(* CODESYS project Exp_1.project
   Company: ifm electronic
   Description: Project template with CR711S configured 2.25MByte Standard 2.25MByte Safety
   Title: ifmCR711S_TemplateProject
   Version: 2.4.10.0

Project tree, tasks and I/O mapping:
  SafetyPLC : CR711S SIL2, ifm electronic, order no. CR711S, version 3.2.0.0
    application Application
      libraries: ifmR360-3, * (ifm electronic)
      task Task (cyclic, interval t#10ms, priority 1, watchdog t#8ms x 1) calls PLC_PRG
      global variables EVL
      program PLC_PRG [ST]
    Communication : Communication, ifm electronic, version 3.2.0.0
      CAN : CAN, ifm electronic, version 3.2.0.0
      Ethernet : Ethernet, ifm electronic, version 3.2.0.0
    HMI : HMI, ifm electronic, version 3.2.0.0
      User_LEDs : User_LEDs, ifm electronic, version 3.2.0.0
          input  UserLED0_I : LED_IEC_B_INPUT_MAPPING_TYPE  // UserLED0_I
          input  UserLED1_I : LED_IEC_B_INPUT_MAPPING_TYPE  // UserLED1_I
          input  UserLED2_I : LED_IEC_B_INPUT_MAPPING_TYPE  // UserLED2_I
          input  UserLED3_I : LED_IEC_B_INPUT_MAPPING_TYPE  // UserLED3_I
          output UserLED0_Q : LED_IEC_B_OUTPUT_MAPPING_TYPE  // User LED 0
          output UserLED1_Q : LED_IEC_B_OUTPUT_MAPPING_TYPE  // User LED 1
          output UserLED2_Q : LED_IEC_B_OUTPUT_MAPPING_TYPE  // User LED 2
          output UserLED3_Q : LED_IEC_B_OUTPUT_MAPPING_TYPE  // User LED 3
    Local_IO : Local_IO, ifm electronic, version 3.2.0.0
      Inputs : Inputs, ifm electronic, version 3.2.0.0
          input  IN0100_I : IN_MULTIFUNCTION_A_INPUT_MAPPING_TYPE  // IN0100_I
          input  IN0101_I : IN_MULTIFUNCTION_A_INPUT_MAPPING_TYPE  // IN0101_I
          input  IN0102_I : IN_MULTIFUNCTION_A_INPUT_MAPPING_TYPE  // IN0102_I
          input  IN0103_I : IN_MULTIFUNCTION_A_INPUT_MAPPING_TYPE  // IN0103_I
          input  IN0200_I : IN_MULTIFUNCTION_A_INPUT_MAPPING_TYPE  // IN0200_I
          input  IN0201_I : IN_MULTIFUNCTION_A_INPUT_MAPPING_TYPE  // IN0201_I
          input  IN0202_I : IN_MULTIFUNCTION_A_INPUT_MAPPING_TYPE  // IN0202_I
          input  IN0203_I : IN_MULTIFUNCTION_A_INPUT_MAPPING_TYPE  // IN0203_I
          input  IN0600_I : IN_MULTIFUNCTION_A_INPUT_MAPPING_TYPE  // IN0600_I
          input  IN0601_I : IN_MULTIFUNCTION_A_INPUT_MAPPING_TYPE  // IN0601_I
          input  IN0602_I : IN_MULTIFUNCTION_A_INPUT_MAPPING_TYPE  // IN0602_I
          input  IN0603_I : IN_MULTIFUNCTION_A_INPUT_MAPPING_TYPE  // IN0603_I
          input  IN0700_I : IN_MULTIFUNCTION_A_INPUT_MAPPING_TYPE  // IN0700_I
          input  IN0701_I : IN_MULTIFUNCTION_A_INPUT_MAPPING_TYPE  // IN0701_I
          input  IN0702_I : IN_MULTIFUNCTION_A_INPUT_MAPPING_TYPE  // IN0702_I
          input  IN0703_I : IN_MULTIFUNCTION_A_INPUT_MAPPING_TYPE  // IN0703_I
          input  IN0400_I : IN_RESISTOR_A_INPUT_MAPPING_TYPE  // IN0400_I
          input  IN0401_I : IN_RESISTOR_A_INPUT_MAPPING_TYPE  // IN0401_I
          input  IN0900_I : IN_RESISTOR_A_INPUT_MAPPING_TYPE  // IN0900_I
          input  IN0901_I : IN_RESISTOR_A_INPUT_MAPPING_TYPE  // IN0901_I
          input  IN0300_I : IN_DIGITAL_B_INPUT_MAPPING_TYPE  // IN0300_I
          input  IN0301_I : IN_DIGITAL_B_INPUT_MAPPING_TYPE  // IN0301_I
          input  IN0800_I : IN_DIGITAL_B_INPUT_MAPPING_TYPE  // IN0800_I
          input  IN0801_I : IN_DIGITAL_B_INPUT_MAPPING_TYPE  // IN0801_I
          input  COM_RESET_I : IN_COMMUNICATION_RESET_INPUT_MAPPING_TYPE  // COM_RESET_I
          input  IN0000_I : IN_FREQUENCY_B_CHANNEL_A_INPUT_MAPPING_TYPE  // IN0000_I
          input  IN0002_I : IN_FREQUENCY_B_CHANNEL_A_INPUT_MAPPING_TYPE  // IN0002_I
          input  IN0500_I : IN_FREQUENCY_B_CHANNEL_A_INPUT_MAPPING_TYPE  // IN0500_I
          input  IN0502_I : IN_FREQUENCY_B_CHANNEL_A_INPUT_MAPPING_TYPE  // IN0502_I
          input  IN0001_I : IN_FREQUENCY_B_CHANNEL_B_INPUT_MAPPING_TYPE  // IN0001_I
          input  IN0003_I : IN_FREQUENCY_B_CHANNEL_B_INPUT_MAPPING_TYPE  // IN0003_I
          input  IN0501_I : IN_FREQUENCY_B_CHANNEL_B_INPUT_MAPPING_TYPE  // IN0501_I
          input  IN0503_I : IN_FREQUENCY_B_CHANNEL_B_INPUT_MAPPING_TYPE  // IN0503_I
      Outputs : Outputs, ifm electronic, version 3.2.0.0
          input  OUT0006_I : OUT_PWM_40_BRIDGE_A_INPUT_MAPPING_TYPE  // OUT0006_I
          input  OUT0106_I : OUT_PWM_40_BRIDGE_A_INPUT_MAPPING_TYPE  // OUT0106_I
          input  OUT0206_I : OUT_PWM_40_BRIDGE_A_INPUT_MAPPING_TYPE  // OUT0206_I
          input  OUT0008_I : OUT_PWM_40_A_INPUT_MAPPING_TYPE  // OUT0008_I
          input  OUT0108_I : OUT_PWM_40_A_INPUT_MAPPING_TYPE  // OUT0108_I
          input  OUT0208_I : OUT_PWM_40_A_INPUT_MAPPING_TYPE  // OUT0208_I
          input  OUT0000_I : OUT_PWM_25_A_INPUT_MAPPING_TYPE  // OUT0000_I
          input  OUT0002_I : OUT_PWM_25_A_INPUT_MAPPING_TYPE  // OUT0002_I
          input  OUT0004_I : OUT_PWM_25_A_INPUT_MAPPING_TYPE  // OUT0004_I
          input  OUT0100_I : OUT_PWM_25_A_INPUT_MAPPING_TYPE  // OUT0100_I
          input  OUT0102_I : OUT_PWM_25_A_INPUT_MAPPING_TYPE  // OUT0102_I
          input  OUT0104_I : OUT_PWM_25_A_INPUT_MAPPING_TYPE  // OUT0104_I
          input  OUT0200_I : OUT_PWM_25_A_INPUT_MAPPING_TYPE  // OUT0200_I
          input  OUT0202_I : OUT_PWM_25_A_INPUT_MAPPING_TYPE  // OUT0202_I
          input  OUT0204_I : OUT_PWM_25_A_INPUT_MAPPING_TYPE  // OUT0204_I
          input  OUT3001_I : OUT_VOLTAGE_A_INPUT_MAPPING_TYPE  // OUT3001_I
          input  OUT3000_I : OUT_SUPPLY_A_INPUT_MAPPING_TYPE  // OUT3000_I
          input  OUT0001_I : OUT_PWM_25_B_INPUT_MAPPING_TYPE  // OUT0001_I
          input  OUT0003_I : OUT_PWM_25_B_INPUT_MAPPING_TYPE  // OUT0003_I
          input  OUT0005_I : OUT_PWM_25_B_INPUT_MAPPING_TYPE  // OUT0005_I
          input  OUT0101_I : OUT_PWM_25_B_INPUT_MAPPING_TYPE  // OUT0101_I
          input  OUT0103_I : OUT_PWM_25_B_INPUT_MAPPING_TYPE  // OUT0103_I
          input  OUT0105_I : OUT_PWM_25_B_INPUT_MAPPING_TYPE  // OUT0105_I
          input  OUT0201_I : OUT_PWM_25_B_INPUT_MAPPING_TYPE  // OUT0201_I
          input  OUT0203_I : OUT_PWM_25_B_INPUT_MAPPING_TYPE  // OUT0203_I
          input  OUT0205_I : OUT_PWM_25_B_INPUT_MAPPING_TYPE  // OUT0205_I
          input  OUT0007_I : OUT_PWM_40_BRIDGE_A_INPUT_MAPPING_TYPE  // OUT0007_I
          input  OUT0107_I : OUT_PWM_40_BRIDGE_A_INPUT_MAPPING_TYPE  // OUT0107_I
          input  OUT0207_I : OUT_PWM_40_BRIDGE_A_INPUT_MAPPING_TYPE  // OUT0207_I
          output OUT0006_Q : OUT_PWM_40_BRIDGE_A_OUTPUT_MAPPING_TYPE  // OUT0006_Q
          output OUT0106_Q : OUT_PWM_40_BRIDGE_A_OUTPUT_MAPPING_TYPE  // OUT0106_Q
          output OUT0206_Q : OUT_PWM_40_BRIDGE_A_OUTPUT_MAPPING_TYPE  // OUT0206_Q
          output OUT0008_Q : OUT_PWM_40_A_OUTPUT_MAPPING_TYPE  // OUT0008_Q
          output OUT0108_Q : OUT_PWM_40_A_OUTPUT_MAPPING_TYPE  // OUT0108_Q
          output OUT0208_Q : OUT_PWM_40_A_OUTPUT_MAPPING_TYPE  // OUT0208_Q
          output OUT0000_Q : OUT_PWM_25_A_OUTPUT_MAPPING_TYPE  // OUT0000_Q
          output OUT0002_Q : OUT_PWM_25_A_OUTPUT_MAPPING_TYPE  // OUT0002_Q
          output OUT0004_Q : OUT_PWM_25_A_OUTPUT_MAPPING_TYPE  // OUT0004_Q
          output OUT0100_Q : OUT_PWM_25_A_OUTPUT_MAPPING_TYPE  // OUT0100_Q
          output OUT0102_Q : OUT_PWM_25_A_OUTPUT_MAPPING_TYPE  // OUT0102_Q
          output OUT0104_Q : OUT_PWM_25_A_OUTPUT_MAPPING_TYPE  // OUT0104_Q
          output OUT0200_Q : OUT_PWM_25_A_OUTPUT_MAPPING_TYPE  // OUT0200_Q
          output OUT0202_Q : OUT_PWM_25_A_OUTPUT_MAPPING_TYPE  // OUT0202_Q
          output OUT0204_Q : OUT_PWM_25_A_OUTPUT_MAPPING_TYPE  // OUT0204_Q
          output OUT3001_Q : OUT_VOLTAGE_A_OUTPUT_MAPPING_TYPE  // OUT3001_Q
          output OUT3000_Q : OUT_SUPPLY_A_OUTPUT_MAPPING_TYPE  // OUT3000_Q
          output OUT0001_Q : OUT_PWM_25_B_OUTPUT_MAPPING_TYPE  // OUT0001_Q
          output OUT0003_Q : OUT_PWM_25_B_OUTPUT_MAPPING_TYPE  // OUT0003_Q
          output OUT0005_Q : OUT_PWM_25_B_OUTPUT_MAPPING_TYPE  // OUT0005_Q
          output OUT0101_Q : OUT_PWM_25_B_OUTPUT_MAPPING_TYPE  // OUT0101_Q
          output OUT0103_Q : OUT_PWM_25_B_OUTPUT_MAPPING_TYPE  // OUT0103_Q
          output OUT0105_Q : OUT_PWM_25_B_OUTPUT_MAPPING_TYPE  // OUT0105_Q
          output OUT0201_Q : OUT_PWM_25_B_OUTPUT_MAPPING_TYPE  // OUT0201_Q
          output OUT0203_Q : OUT_PWM_25_B_OUTPUT_MAPPING_TYPE  // OUT0203_Q
          output OUT0205_Q : OUT_PWM_25_B_OUTPUT_MAPPING_TYPE  // OUT0205_Q
          output OUT0007_Q : OUT_PWM_40_BRIDGE_A_OUTPUT_MAPPING_TYPE  // OUT0007_Q
          output OUT0107_Q : OUT_PWM_40_BRIDGE_A_OUTPUT_MAPPING_TYPE  // OUT0107_Q
          output OUT0207_Q : OUT_PWM_40_BRIDGE_A_OUTPUT_MAPPING_TYPE  // OUT0207_Q
      System_Inputs : System_Inputs, ifm electronic, version 3.2.0.0
          input  VBB30 : IN_SYSTEM_VOLTAGE_INPUT_MAPPING_TYPE  // VBB30
          input  VBB15 : IN_SYSTEM_VOLTAGE_INPUT_MAPPING_TYPE  // VBB15
          input  TemperatureBoard0 : IN_TEMPERATURE_INPUT_MAPPING_TYPE  // TemperatureBoard0
          input  TemperatureChip0 : IN_TEMPERATURE_INPUT_MAPPING_TYPE  // TemperatureChip0
      System_Outputs : System_Outputs, ifm electronic, version 3.2.0.0
          input  VBB0_SW_I : OUT_GROUP_SWITCH_INPUT_MAPPING_TYPE  // VBB0_SW_I
          input  VBB1_SW_I : OUT_GROUP_SWITCH_INPUT_MAPPING_TYPE  // VBB1_SW_I
          input  VBB2_SW_I : OUT_GROUP_SWITCH_INPUT_MAPPING_TYPE  // VBB2_SW_I
          output VBB0_SW_Q : OUT_GROUP_SWITCH_OUTPUT_MAPPING_TYPE  // VBB0_SW_Q
          output VBB1_SW_Q : OUT_GROUP_SWITCH_OUTPUT_MAPPING_TYPE  // VBB1_SW_Q
          output VBB2_SW_Q : OUT_GROUP_SWITCH_OUTPUT_MAPPING_TYPE  // VBB2_SW_Q
          output SUPPLY_SWITCH_Q : OUT_SYS_SWITCH_OUTPUT_MAPPING_TYPE  // SUPPLY_SWITCH_Q
  StandardPLC : CR711S Standard, ifm electronic, order no. CR711S, version 3.2.0.0
    application Application
      libraries: ifmR360-3, 1.1.1.0 (ifm electronic); Util, * (System); Standard, * (System); CR711S IOWrapper, 1.0.4.9 (ifm electronic)
      task Task (cyclic, interval t#10ms, priority 0) calls PLC_PRG
      EVC
      program PLC_PRG [ST]
      program CR711S_Config [ST]: config_inputs, config_outgroups, config_outputs
      program CAN_INIT [ST]
      program CA_TX [FBD]
      program CAN_RX [FBD]
    Communication : Communication, ifm electronic, version 3.2.0.0
      CAN : CAN, ifm electronic, version 3.2.0.0
      Ethernet : Ethernet, ifm electronic, version 3.2.0.0
    HMI : HMI, ifm electronic, version 3.2.0.0
      User_LEDs : User_LEDs, ifm electronic, version 3.2.0.0
          input  UserLED0_I : LED_IEC_B_INPUT_MAPPING_TYPE  // UserLED0_I
          input  UserLED1_I : LED_IEC_B_INPUT_MAPPING_TYPE  // UserLED1_I
          input  UserLED2_I : LED_IEC_B_INPUT_MAPPING_TYPE  // UserLED2_I
          input  UserLED3_I : LED_IEC_B_INPUT_MAPPING_TYPE  // UserLED3_I
          output UserLED0_Q : LED_IEC_B_OUTPUT_MAPPING_TYPE  // User LED 0
          output UserLED1_Q : LED_IEC_B_OUTPUT_MAPPING_TYPE  // User LED 1
          output UserLED2_Q : LED_IEC_B_OUTPUT_MAPPING_TYPE  // User LED 2
          output UserLED3_Q : LED_IEC_B_OUTPUT_MAPPING_TYPE  // User LED 3
    Local_IO : Local_IO, ifm electronic, version 3.2.0.0
      Inputs : Inputs, ifm electronic, version 3.2.0.0
          input  IN0100_I : IN_MULTIFUNCTION_A_INPUT_MAPPING_TYPE  // IN0100_I
          input  IN0101_I : IN_MULTIFUNCTION_A_INPUT_MAPPING_TYPE  // IN0101_I
          input  IN0102_I : IN_MULTIFUNCTION_A_INPUT_MAPPING_TYPE  // IN0102_I
          input  IN0103_I : IN_MULTIFUNCTION_A_INPUT_MAPPING_TYPE  // IN0103_I
          input  IN0200_I : IN_MULTIFUNCTION_A_INPUT_MAPPING_TYPE  // IN0200_I
          input  IN0201_I : IN_MULTIFUNCTION_A_INPUT_MAPPING_TYPE  // IN0201_I
          input  IN0202_I : IN_MULTIFUNCTION_A_INPUT_MAPPING_TYPE  // IN0202_I
          input  IN0203_I : IN_MULTIFUNCTION_A_INPUT_MAPPING_TYPE  // IN0203_I
          input  IN0600_I : IN_MULTIFUNCTION_A_INPUT_MAPPING_TYPE  // IN0600_I
          input  IN0601_I : IN_MULTIFUNCTION_A_INPUT_MAPPING_TYPE  // IN0601_I
          input  IN0602_I : IN_MULTIFUNCTION_A_INPUT_MAPPING_TYPE  // IN0602_I
          input  IN0603_I : IN_MULTIFUNCTION_A_INPUT_MAPPING_TYPE  // IN0603_I
          input  IN0700_I : IN_MULTIFUNCTION_A_INPUT_MAPPING_TYPE  // IN0700_I
          input  IN0701_I : IN_MULTIFUNCTION_A_INPUT_MAPPING_TYPE  // IN0701_I
          input  IN0702_I : IN_MULTIFUNCTION_A_INPUT_MAPPING_TYPE  // IN0702_I
          input  IN0703_I : IN_MULTIFUNCTION_A_INPUT_MAPPING_TYPE  // IN0703_I
          input  IN0400_I : IN_RESISTOR_A_INPUT_MAPPING_TYPE  // IN0400_I
          input  IN0401_I : IN_RESISTOR_A_INPUT_MAPPING_TYPE  // IN0401_I
          input  IN0900_I : IN_RESISTOR_A_INPUT_MAPPING_TYPE  // IN0900_I
          input  IN0901_I : IN_RESISTOR_A_INPUT_MAPPING_TYPE  // IN0901_I
          input  IN0300_I : IN_DIGITAL_B_INPUT_MAPPING_TYPE  // IN0300_I
          input  IN0301_I : IN_DIGITAL_B_INPUT_MAPPING_TYPE  // IN0301_I
          input  IN0800_I : IN_DIGITAL_B_INPUT_MAPPING_TYPE  // IN0800_I
          input  IN0801_I : IN_DIGITAL_B_INPUT_MAPPING_TYPE  // IN0801_I
          input  COM_RESET_I : IN_COMMUNICATION_RESET_INPUT_MAPPING_TYPE  // COM_RESET_I
          input  IN0000_I : IN_FREQUENCY_B_CHANNEL_A_INPUT_MAPPING_TYPE  // IN0000_I
          input  IN0002_I : IN_FREQUENCY_B_CHANNEL_A_INPUT_MAPPING_TYPE  // IN0002_I
          input  IN0500_I : IN_FREQUENCY_B_CHANNEL_A_INPUT_MAPPING_TYPE  // IN0500_I
          input  IN0502_I : IN_FREQUENCY_B_CHANNEL_A_INPUT_MAPPING_TYPE  // IN0502_I
          input  IN0001_I : IN_FREQUENCY_B_CHANNEL_B_INPUT_MAPPING_TYPE  // IN0001_I
          input  IN0003_I : IN_FREQUENCY_B_CHANNEL_B_INPUT_MAPPING_TYPE  // IN0003_I
          input  IN0501_I : IN_FREQUENCY_B_CHANNEL_B_INPUT_MAPPING_TYPE  // IN0501_I
          input  IN0503_I : IN_FREQUENCY_B_CHANNEL_B_INPUT_MAPPING_TYPE  // IN0503_I
      Outputs : Outputs, ifm electronic, version 3.2.0.0
          input  OUT0006_I : OUT_PWM_40_BRIDGE_A_INPUT_MAPPING_TYPE  // OUT0006_I
          input  OUT0106_I : OUT_PWM_40_BRIDGE_A_INPUT_MAPPING_TYPE  // OUT0106_I
          input  OUT0206_I : OUT_PWM_40_BRIDGE_A_INPUT_MAPPING_TYPE  // OUT0206_I
          input  OUT0008_I : OUT_PWM_40_A_INPUT_MAPPING_TYPE  // OUT0008_I
          input  OUT0108_I : OUT_PWM_40_A_INPUT_MAPPING_TYPE  // OUT0108_I
          input  OUT0208_I : OUT_PWM_40_A_INPUT_MAPPING_TYPE  // OUT0208_I
          input  OUT0000_I : OUT_PWM_25_A_INPUT_MAPPING_TYPE  // OUT0000_I
          input  OUT0002_I : OUT_PWM_25_A_INPUT_MAPPING_TYPE  // OUT0002_I
          input  OUT0004_I : OUT_PWM_25_A_INPUT_MAPPING_TYPE  // OUT0004_I
          input  OUT0100_I : OUT_PWM_25_A_INPUT_MAPPING_TYPE  // OUT0100_I
          input  OUT0102_I : OUT_PWM_25_A_INPUT_MAPPING_TYPE  // OUT0102_I
          input  OUT0104_I : OUT_PWM_25_A_INPUT_MAPPING_TYPE  // OUT0104_I
          input  OUT0200_I : OUT_PWM_25_A_INPUT_MAPPING_TYPE  // OUT0200_I
          input  OUT0202_I : OUT_PWM_25_A_INPUT_MAPPING_TYPE  // OUT0202_I
          input  OUT0204_I : OUT_PWM_25_A_INPUT_MAPPING_TYPE  // OUT0204_I
          input  OUT3001_I : OUT_VOLTAGE_A_INPUT_MAPPING_TYPE  // OUT3001_I
          input  OUT3000_I : OUT_SUPPLY_A_INPUT_MAPPING_TYPE  // OUT3000_I
          input  OUT0001_I : OUT_PWM_25_B_INPUT_MAPPING_TYPE  // OUT0001_I
          input  OUT0003_I : OUT_PWM_25_B_INPUT_MAPPING_TYPE  // OUT0003_I
          input  OUT0005_I : OUT_PWM_25_B_INPUT_MAPPING_TYPE  // OUT0005_I
          input  OUT0101_I : OUT_PWM_25_B_INPUT_MAPPING_TYPE  // OUT0101_I
          input  OUT0103_I : OUT_PWM_25_B_INPUT_MAPPING_TYPE  // OUT0103_I
          input  OUT0105_I : OUT_PWM_25_B_INPUT_MAPPING_TYPE  // OUT0105_I
          input  OUT0201_I : OUT_PWM_25_B_INPUT_MAPPING_TYPE  // OUT0201_I
          input  OUT0203_I : OUT_PWM_25_B_INPUT_MAPPING_TYPE  // OUT0203_I
          input  OUT0205_I : OUT_PWM_25_B_INPUT_MAPPING_TYPE  // OUT0205_I
          input  OUT0007_I : OUT_PWM_40_BRIDGE_A_INPUT_MAPPING_TYPE  // OUT0007_I
          input  OUT0107_I : OUT_PWM_40_BRIDGE_A_INPUT_MAPPING_TYPE  // OUT0107_I
          input  OUT0207_I : OUT_PWM_40_BRIDGE_A_INPUT_MAPPING_TYPE  // OUT0207_I
          output OUT0006_Q : OUT_PWM_40_BRIDGE_A_OUTPUT_MAPPING_TYPE  // OUT0006_Q
          output OUT0106_Q : OUT_PWM_40_BRIDGE_A_OUTPUT_MAPPING_TYPE  // OUT0106_Q
          output OUT0206_Q : OUT_PWM_40_BRIDGE_A_OUTPUT_MAPPING_TYPE  // OUT0206_Q
          output OUT0008_Q : OUT_PWM_40_A_OUTPUT_MAPPING_TYPE  // OUT0008_Q
          output OUT0108_Q : OUT_PWM_40_A_OUTPUT_MAPPING_TYPE  // OUT0108_Q
          output OUT0208_Q : OUT_PWM_40_A_OUTPUT_MAPPING_TYPE  // OUT0208_Q
          output OUT0000_Q : OUT_PWM_25_A_OUTPUT_MAPPING_TYPE  // OUT0000_Q
          output OUT0002_Q : OUT_PWM_25_A_OUTPUT_MAPPING_TYPE  // OUT0002_Q
          output OUT0004_Q : OUT_PWM_25_A_OUTPUT_MAPPING_TYPE  // OUT0004_Q
          output OUT0100_Q : OUT_PWM_25_A_OUTPUT_MAPPING_TYPE  // OUT0100_Q
          output OUT0102_Q : OUT_PWM_25_A_OUTPUT_MAPPING_TYPE  // OUT0102_Q
          output OUT0104_Q : OUT_PWM_25_A_OUTPUT_MAPPING_TYPE  // OUT0104_Q
          output OUT0200_Q : OUT_PWM_25_A_OUTPUT_MAPPING_TYPE  // OUT0200_Q
          output OUT0202_Q : OUT_PWM_25_A_OUTPUT_MAPPING_TYPE  // OUT0202_Q
          output OUT0204_Q : OUT_PWM_25_A_OUTPUT_MAPPING_TYPE  // OUT0204_Q
          output OUT3001_Q : OUT_VOLTAGE_A_OUTPUT_MAPPING_TYPE  // OUT3001_Q
          output OUT3000_Q : OUT_SUPPLY_A_OUTPUT_MAPPING_TYPE  // OUT3000_Q
          output OUT0001_Q : OUT_PWM_25_B_OUTPUT_MAPPING_TYPE  // OUT0001_Q
          output OUT0003_Q : OUT_PWM_25_B_OUTPUT_MAPPING_TYPE  // OUT0003_Q
          output OUT0005_Q : OUT_PWM_25_B_OUTPUT_MAPPING_TYPE  // OUT0005_Q
          output OUT0101_Q : OUT_PWM_25_B_OUTPUT_MAPPING_TYPE  // OUT0101_Q
          output OUT0103_Q : OUT_PWM_25_B_OUTPUT_MAPPING_TYPE  // OUT0103_Q
          output OUT0105_Q : OUT_PWM_25_B_OUTPUT_MAPPING_TYPE  // OUT0105_Q
          output OUT0201_Q : OUT_PWM_25_B_OUTPUT_MAPPING_TYPE  // OUT0201_Q
          output OUT0203_Q : OUT_PWM_25_B_OUTPUT_MAPPING_TYPE  // OUT0203_Q
          output OUT0205_Q : OUT_PWM_25_B_OUTPUT_MAPPING_TYPE  // OUT0205_Q
          output OUT0007_Q : OUT_PWM_40_BRIDGE_A_OUTPUT_MAPPING_TYPE  // OUT0007_Q
          output OUT0107_Q : OUT_PWM_40_BRIDGE_A_OUTPUT_MAPPING_TYPE  // OUT0107_Q
          output OUT0207_Q : OUT_PWM_40_BRIDGE_A_OUTPUT_MAPPING_TYPE  // OUT0207_Q
      System_Inputs : System_Inputs, ifm electronic, version 3.2.0.0
          input  VBB30 : IN_SYSTEM_VOLTAGE_INPUT_MAPPING_TYPE  // VBB30
          input  VBB15 : IN_SYSTEM_VOLTAGE_INPUT_MAPPING_TYPE  // VBB15
          input  TemperatureBoard0 : IN_TEMPERATURE_INPUT_MAPPING_TYPE  // TemperatureBoard0
          input  TemperatureChip0 : IN_TEMPERATURE_INPUT_MAPPING_TYPE  // TemperatureChip0
      System_Outputs : System_Outputs, ifm electronic, version 3.2.0.0
          input  VBB0_SW_I : OUT_GROUP_SWITCH_INPUT_MAPPING_TYPE  // VBB0_SW_I
          input  VBB1_SW_I : OUT_GROUP_SWITCH_INPUT_MAPPING_TYPE  // VBB1_SW_I
          input  VBB2_SW_I : OUT_GROUP_SWITCH_INPUT_MAPPING_TYPE  // VBB2_SW_I
          output VBB0_SW_Q : OUT_GROUP_SWITCH_OUTPUT_MAPPING_TYPE  // VBB0_SW_Q
          output VBB1_SW_Q : OUT_GROUP_SWITCH_OUTPUT_MAPPING_TYPE  // VBB1_SW_Q
          output VBB2_SW_Q : OUT_GROUP_SWITCH_OUTPUT_MAPPING_TYPE  // VBB2_SW_Q
          output SUPPLY_SWITCH_Q : OUT_SYS_SWITCH_OUTPUT_MAPPING_TYPE  // SUPPLY_SWITCH_Q
  CR711S : CR711S, ifm electronic, order no. CR711S, version 3.2.0.0
*)

// SafetyPLC/Application/EVL
(* THIS EVL IS AUTOGENERATED. DO NOT MODIFY THESE ATTRIBUTES. *)
{attribute 'location' := '16#800' }
{attribute 'linkalways'}
{attribute 'qualified_only'}
VAR_GLOBAL

END_VAR

// SafetyPLC/Application/PLC_PRG
PROGRAM PLC_PRG
VAR

END_VAR

END_PROGRAM

// StandardPLC/Application/PLC_PRG
PROGRAM PLC_PRG
VAR
	CA_RX: INT;
END_VAR
(*
IOWrapper V1.0.4.4
ifm ecomatic gmbh - VNC - pp 

The licence free software is of average quality and suitable for normal use on common personal
computers. According to the present state of software technology no guarantee can be
assumed for the correct operation or absence of computer viruses nor for the removal of any
fault which may occur. In case of an incorrect program ifm electronic gmbh cannot be held
liable for cost incurred at the customer (e.g. maintenance, repair or rectification of faults).
The exclusion does not apply to damage for which liability is mandatory according to peremptory
legal provisions. Copyright by ifm electronic gmbh, Essen. No copies may be made without the
written permission of ifm electronic gmbh. This also goes for printing images or text for business
use. We reserve the right to make technical alterations.
*)

CR711S_Config(); 			//IO Configuration

IOWrapper.READ_INPUTS(); 	//Call IOWrapper Main Program and Read Data from Inputs   
CAN_INIT();
CA_TX();
CAN_RX();


							//Put your Application program here 

IOWrapper.WRITE_OUTPUTS();	//Call IOWrapper Main Program and Write Data to Outputs

END_PROGRAM

// StandardPLC/Application/CR711S_Config
PROGRAM CR711S_Config
VAR_INPUT
END_VAR
(*
IOWrapper V1.4.2.3
ifm ecomatic - VNC - pp 

The licence free software is of average quality and suitable for normal use on common personal
computers. According to the present state of software technology no guarantee can be
assumed for the correct operation or absence of computer viruses nor for the removal of any
fault which may occur. In case of an incorrect program ifm electronic gmbh cannot be held
liable for cost incurred at the customer (e.g. maintenance, repair or rectification of faults).
The exclusion does not apply to damage for which liability is mandatory according to peremptory
legal provisions. Copyright by ifm electronic gmbh, Essen. No copies may be made without the
written permission of ifm electronic gmbh. This also goes for printing images or text for business
use. We reserve the right to make technical alterations.
*)

(* IO Configuration*)
config_inputs();
config_outputs();
config_outgroups();

ACTION config_inputs:
(* Input Mode Configuration *) // FREQ_SENSE_PERIODS.PERIODS_5, ENCODER_RESOLUTION.EVERY_EDGE
(* Frequency Inputs *)
IN0000.CONFIG.MONITOR		(FILTER_INPUT.UNCHANGED);
IN0001.CONFIG.MONITOR		(FILTER_INPUT.UNCHANGED);
IN0002.CONFIG.MONITOR		(FILTER_INPUT.UNCHANGED);
IN0003.CONFIG.MONITOR		(FILTER_INPUT.UNCHANGED);
IN0500.CONFIG.MONITOR		(FILTER_INPUT.UNCHANGED);
IN0501.CONFIG.MONITOR		(FILTER_INPUT.UNCHANGED);
IN0502.CONFIG.MONITOR		(FILTER_INPUT.UNCHANGED);
IN0503.CONFIG.MONITOR		(FILTER_INPUT.UNCHANGED);
(* Multifuntional Inputs *) 
IN0100.CONFIG.MONITOR		(FILTER_INPUT.UNCHANGED);
IN0101.CONFIG.MONITOR		(FILTER_INPUT.UNCHANGED);
IN0102.CONFIG.MONITOR		(FILTER_INPUT.UNCHANGED);
IN0103.CONFIG.MONITOR		(FILTER_INPUT.UNCHANGED);
IN0200.CONFIG.MONITOR		(FILTER_INPUT.UNCHANGED);
IN0201.CONFIG.MONITOR		(FILTER_INPUT.UNCHANGED);
IN0202.CONFIG.MONITOR		(FILTER_INPUT.UNCHANGED);
IN0203.CONFIG.MONITOR		(FILTER_INPUT.UNCHANGED);
                  				
IN0600.CONFIG.MONITOR		(FILTER_INPUT.UNCHANGED);
IN0601.CONFIG.MONITOR		(FILTER_INPUT.UNCHANGED);
IN0602.CONFIG.MONITOR		(FILTER_INPUT.UNCHANGED);
IN0603.CONFIG.MONITOR		(FILTER_INPUT.UNCHANGED);
IN0700.CONFIG.MONITOR		(FILTER_INPUT.UNCHANGED);
IN0701.CONFIG.MONITOR		(FILTER_INPUT.UNCHANGED);
IN0702.CONFIG.MONITOR		(FILTER_INPUT.UNCHANGED);
IN0703.CONFIG.MONITOR		(FILTER_INPUT.UNCHANGED);
(* Digital Inputs *) 				
IN0300.CONFIG.MONITOR		(FILTER_INPUT.UNCHANGED);
IN0301.CONFIG.MONITOR		(FILTER_INPUT.UNCHANGED);
IN0800.CONFIG.MONITOR		(FILTER_INPUT.UNCHANGED);
IN0801.CONFIG.MONITOR		(FILTER_INPUT.UNCHANGED);
(* Resistopr Inputs *)      	
IN0400.CONFIG.MONITOR		(FILTER_INPUT.UNCHANGED);
IN0401.CONFIG.MONITOR		(FILTER_INPUT.UNCHANGED);
IN0900.CONFIG.MONITOR		(FILTER_INPUT.UNCHANGED);
IN0901.CONFIG.MONITOR		(FILTER_INPUT.UNCHANGED);

(* Diagnostic and Protection Configuration *) //eDIAG_PROT_MODE.DIAG_PROT
(* Frequency Inputs *) 
IN0000.CONFIG.SET_DIAG_LVL_PROT		(0, 32000, 100, eDIAG_PROT_MODE.DIAG_PROT);
IN0001.CONFIG.SET_DIAG_LVL_PROT		(0, 32000, 100, eDIAG_PROT_MODE.DIAG_PROT);
IN0002.CONFIG.SET_DIAG_LVL_PROT		(0, 32000, 100, eDIAG_PROT_MODE.DIAG_PROT);
IN0003.CONFIG.SET_DIAG_LVL_PROT		(0, 32000, 100, eDIAG_PROT_MODE.DIAG_PROT);
IN0500.CONFIG.SET_DIAG_LVL_PROT		(0, 32000, 100, eDIAG_PROT_MODE.DIAG_PROT);
IN0501.CONFIG.SET_DIAG_LVL_PROT		(0, 32000, 100, eDIAG_PROT_MODE.DIAG_PROT);
IN0502.CONFIG.SET_DIAG_LVL_PROT		(0, 32000, 100, eDIAG_PROT_MODE.DIAG_PROT);
IN0503.CONFIG.SET_DIAG_LVL_PROT		(0, 32000, 100, eDIAG_PROT_MODE.DIAG_PROT);
(* Multifuntional Inputs *)                          
IN0100.CONFIG.SET_DIAG_LVL_PROT		(0, 32000, 100, eDIAG_PROT_MODE.DIAG_PROT);
IN0101.CONFIG.SET_DIAG_LVL_PROT		(0, 32000, 100, eDIAG_PROT_MODE.DIAG_PROT);
IN0102.CONFIG.SET_DIAG_LVL_PROT		(0, 32000, 100, eDIAG_PROT_MODE.DIAG_PROT);
IN0103.CONFIG.SET_DIAG_LVL_PROT		(0, 32000, 100, eDIAG_PROT_MODE.DIAG_PROT);
IN0200.CONFIG.SET_DIAG_LVL_PROT		(0, 32000, 100, eDIAG_PROT_MODE.DIAG_PROT);
IN0201.CONFIG.SET_DIAG_LVL_PROT		(0, 32000, 100, eDIAG_PROT_MODE.DIAG_PROT);
IN0202.CONFIG.SET_DIAG_LVL_PROT		(0, 32000, 100, eDIAG_PROT_MODE.DIAG_PROT);
IN0203.CONFIG.SET_DIAG_LVL_PROT		(0, 32000, 100, eDIAG_PROT_MODE.DIAG_PROT);
                                                     
IN0600.CONFIG.SET_DIAG_LVL_PROT		(0, 32000, 100, eDIAG_PROT_MODE.DIAG_PROT);
IN0601.CONFIG.SET_DIAG_LVL_PROT		(0, 32000, 100, eDIAG_PROT_MODE.DIAG_PROT);
IN0602.CONFIG.SET_DIAG_LVL_PROT		(0, 32000, 100, eDIAG_PROT_MODE.DIAG_PROT);
IN0603.CONFIG.SET_DIAG_LVL_PROT		(0, 32000, 100, eDIAG_PROT_MODE.DIAG_PROT);
IN0700.CONFIG.SET_DIAG_LVL_PROT		(0, 32000, 100, eDIAG_PROT_MODE.DIAG_PROT);
IN0701.CONFIG.SET_DIAG_LVL_PROT		(0, 32000, 100, eDIAG_PROT_MODE.DIAG_PROT);
IN0702.CONFIG.SET_DIAG_LVL_PROT		(0, 32000, 100, eDIAG_PROT_MODE.DIAG_PROT);
IN0703.CONFIG.SET_DIAG_LVL_PROT		(0, 32000, 100, eDIAG_PROT_MODE.DIAG_PROT);
(* Digital Inputs *)                                 
IN0300.CONFIG.SET_DIAG_LVL_PROT		(0, 32000, 100, eDIAG_PROT_MODE.DIAG_PROT);
IN0301.CONFIG.SET_DIAG_LVL_PROT		(0, 32000, 100, eDIAG_PROT_MODE.DIAG_PROT);
IN0800.CONFIG.SET_DIAG_LVL_PROT		(0, 32000, 100, eDIAG_PROT_MODE.DIAG_PROT);
IN0801.CONFIG.SET_DIAG_LVL_PROT		(0, 32000, 100, eDIAG_PROT_MODE.DIAG_PROT);
(* Resistopr Inputs *)                               
IN0400.CONFIG.SET_DIAG_LVL_PROT		(0, 32000, 100, eDIAG_PROT_MODE.DIAG_PROT);
IN0401.CONFIG.SET_DIAG_LVL_PROT		(0, 32000, 100, eDIAG_PROT_MODE.DIAG_PROT);
IN0900.CONFIG.SET_DIAG_LVL_PROT		(0, 32000, 100, eDIAG_PROT_MODE.DIAG_PROT);
IN0901.CONFIG.SET_DIAG_LVL_PROT		(0, 32000, 100, eDIAG_PROT_MODE.DIAG_PROT);

(* Digital Switching Threshold - Default ON:= 0.7*Vbb, OFF:= 0.3*Vbb *)
(* Frequency Inputs *)
IN0000.CONFIG.SET_SWITCH_THRESHOLD(300, 700);
IN0001.CONFIG.SET_SWITCH_THRESHOLD(300, 700);
IN0002.CONFIG.SET_SWITCH_THRESHOLD(300, 700);
IN0003.CONFIG.SET_SWITCH_THRESHOLD(300, 700);
IN0500.CONFIG.SET_SWITCH_THRESHOLD(300, 700);
IN0501.CONFIG.SET_SWITCH_THRESHOLD(300, 700);
IN0502.CONFIG.SET_SWITCH_THRESHOLD(300, 700);
IN0503.CONFIG.SET_SWITCH_THRESHOLD(300, 700);
(* Multifuntional Inputs *) 
IN0100.CONFIG.SET_SWITCH_THRESHOLD(300, 700);
IN0101.CONFIG.SET_SWITCH_THRESHOLD(300, 700);
IN0102.CONFIG.SET_SWITCH_THRESHOLD(300, 700);
IN0103.CONFIG.SET_SWITCH_THRESHOLD(300, 700);
IN0200.CONFIG.SET_SWITCH_THRESHOLD(300, 700);
IN0201.CONFIG.SET_SWITCH_THRESHOLD(300, 700);
IN0202.CONFIG.SET_SWITCH_THRESHOLD(300, 700);
IN0203.CONFIG.SET_SWITCH_THRESHOLD(300, 700);
      
IN0600.CONFIG.SET_SWITCH_THRESHOLD(300, 700);
IN0601.CONFIG.SET_SWITCH_THRESHOLD(300, 700);
IN0602.CONFIG.SET_SWITCH_THRESHOLD(300, 700);
IN0603.CONFIG.SET_SWITCH_THRESHOLD(300, 700);
IN0700.CONFIG.SET_SWITCH_THRESHOLD(300, 700);
IN0701.CONFIG.SET_SWITCH_THRESHOLD(300, 700);
IN0702.CONFIG.SET_SWITCH_THRESHOLD(300, 700);
IN0703.CONFIG.SET_SWITCH_THRESHOLD(300, 700);
(* Digital Inputs *)  
IN0300.CONFIG.SET_SWITCH_THRESHOLD(300, 700);
IN0301.CONFIG.SET_SWITCH_THRESHOLD(300, 700);
IN0800.CONFIG.SET_SWITCH_THRESHOLD(300, 700);
IN0801.CONFIG.SET_SWITCH_THRESHOLD(300, 700);
(* Resistopr Inputs *)   
IN0400.CONFIG.SET_SWITCH_THRESHOLD(300, 700);
IN0401.CONFIG.SET_SWITCH_THRESHOLD(300, 700);
IN0900.CONFIG.SET_SWITCH_THRESHOLD(300, 700);
IN0901.CONFIG.SET_SWITCH_THRESHOLD(300, 700);
END_ACTION

ACTION config_outgroups:
(* Output Group Mode Configuration *) 
OUTGROUP0.CONFIG.MONITOR				(FILTER_OUTPUT_GROUP.UNCHANGED);
OUTGROUP1.CONFIG.MONITOR				(FILTER_OUTPUT_GROUP.UNCHANGED);
OUTGROUP2.CONFIG.MONITOR				(FILTER_OUTPUT_GROUP.UNCHANGED);

(* Diagnostic and Protection Configuration *) 
OUTGROUP0.CONFIG.SET_DIAG_LVL_PROT		(0, 12000, 100, eDIAG_PROT_MODE.DIAG_PROT);
OUTGROUP1.CONFIG.SET_DIAG_LVL_PROT		(0, 12000, 100, eDIAG_PROT_MODE.DIAG_PROT);
OUTGROUP2.CONFIG.SET_DIAG_LVL_PROT		(0, 12000, 100, eDIAG_PROT_MODE.DIAG_PROT);
END_ACTION

ACTION config_outputs:
(* Output Mode Configuration *) 
(* Group 0 *)
OUT0000.CONFIG.MONITOR				(FILTER_OUTPUT.UNCHANGED);
OUT0001.CONFIG.MONITOR				(FILTER_OUTPUT.UNCHANGED);
OUT0002.CONFIG.MONITOR				(FILTER_OUTPUT.UNCHANGED);
OUT0003.CONFIG.MONITOR				(FILTER_OUTPUT.UNCHANGED);
OUT0004.CONFIG.MONITOR				(FILTER_OUTPUT.UNCHANGED);
OUT0005.CONFIG.MONITOR				(FILTER_OUTPUT.UNCHANGED);
OUT0006.CONFIG.MONITOR				(FILTER_OUTPUT.UNCHANGED);
OUT0007.CONFIG.MONITOR				(FILTER_OUTPUT.UNCHANGED);
OUT0008.CONFIG.MONITOR				(FILTER_OUTPUT.UNCHANGED);
(* Group 1 *)         				    		
OUT0100.CONFIG.MONITOR				(FILTER_OUTPUT.UNCHANGED);
OUT0101.CONFIG.MONITOR				(FILTER_OUTPUT.UNCHANGED);
OUT0102.CONFIG.MONITOR				(FILTER_OUTPUT.UNCHANGED);
OUT0103.CONFIG.MONITOR				(FILTER_OUTPUT.UNCHANGED);
OUT0104.CONFIG.MONITOR				(FILTER_OUTPUT.UNCHANGED);
OUT0105.CONFIG.MONITOR				(FILTER_OUTPUT.UNCHANGED);
OUT0106.CONFIG.MONITOR				(FILTER_OUTPUT.UNCHANGED);
OUT0107.CONFIG.MONITOR				(FILTER_OUTPUT.UNCHANGED);
OUT0108.CONFIG.MONITOR				(FILTER_OUTPUT.UNCHANGED);
(* Group 2 *)         				    		
OUT0200.CONFIG.MONITOR				(FILTER_OUTPUT.UNCHANGED);
OUT0201.CONFIG.MONITOR				(FILTER_OUTPUT.UNCHANGED);
OUT0202.CONFIG.MONITOR				(FILTER_OUTPUT.UNCHANGED);
OUT0203.CONFIG.MONITOR				(FILTER_OUTPUT.UNCHANGED);
OUT0204.CONFIG.MONITOR				(FILTER_OUTPUT.UNCHANGED);
OUT0205.CONFIG.MONITOR				(FILTER_OUTPUT.UNCHANGED);
OUT0206.CONFIG.MONITOR				(FILTER_OUTPUT.UNCHANGED);
OUT0207.CONFIG.MONITOR				(FILTER_OUTPUT.UNCHANGED);
OUT0208.CONFIG.MONITOR				(FILTER_OUTPUT.UNCHANGED);
(* Output SensorSupply and Analogue *)      				           				
OUT3000.CONFIG.MONITOR				(FILTER_OUTPUT.UNCHANGED);
OUT3001.CONFIG.MONITOR				(FILTER_OUTPUT.UNCHANGED);

(* Diagnostic and Protection Configuration *) 
(* Group 0 *)
OUT0000.CONFIG.SET_DIAG_LVL_PROT	(0, 2500, 100, eDIAG_PROT_MODE.DIAG_PROT);
OUT0001.CONFIG.SET_DIAG_LVL_PROT	(0, 2500, 100, eDIAG_PROT_MODE.DIAG_PROT);
OUT0002.CONFIG.SET_DIAG_LVL_PROT	(0, 2500, 100, eDIAG_PROT_MODE.DIAG_PROT);
OUT0003.CONFIG.SET_DIAG_LVL_PROT	(0, 2500, 100, eDIAG_PROT_MODE.DIAG_PROT);
OUT0004.CONFIG.SET_DIAG_LVL_PROT	(0, 2500, 100, eDIAG_PROT_MODE.DIAG_PROT);
OUT0005.CONFIG.SET_DIAG_LVL_PROT	(0, 2500, 100, eDIAG_PROT_MODE.DIAG_PROT);
OUT0006.CONFIG.SET_DIAG_LVL_PROT	(0, 4000, 100, eDIAG_PROT_MODE.DIAG_PROT);
OUT0007.CONFIG.SET_DIAG_LVL_PROT	(0, 4000, 100, eDIAG_PROT_MODE.DIAG_PROT);
OUT0008.CONFIG.SET_DIAG_LVL_PROT	(0, 4000, 100, eDIAG_PROT_MODE.DIAG_PROT);
(* Group 1 *)                                       
OUT0100.CONFIG.SET_DIAG_LVL_PROT	(0, 2500, 100, eDIAG_PROT_MODE.DIAG_PROT);
OUT0101.CONFIG.SET_DIAG_LVL_PROT	(0, 2500, 100, eDIAG_PROT_MODE.DIAG_PROT);
OUT0102.CONFIG.SET_DIAG_LVL_PROT	(0, 2500, 100, eDIAG_PROT_MODE.DIAG_PROT);
OUT0103.CONFIG.SET_DIAG_LVL_PROT	(0, 2500, 100, eDIAG_PROT_MODE.DIAG_PROT);
OUT0104.CONFIG.SET_DIAG_LVL_PROT	(0, 2500, 100, eDIAG_PROT_MODE.DIAG_PROT);
OUT0105.CONFIG.SET_DIAG_LVL_PROT	(0, 2500, 100, eDIAG_PROT_MODE.DIAG_PROT);
OUT0106.CONFIG.SET_DIAG_LVL_PROT	(0, 4000, 100, eDIAG_PROT_MODE.DIAG_PROT);
OUT0107.CONFIG.SET_DIAG_LVL_PROT	(0, 4000, 100, eDIAG_PROT_MODE.DIAG_PROT);
OUT0108.CONFIG.SET_DIAG_LVL_PROT	(0, 4000, 100, eDIAG_PROT_MODE.DIAG_PROT);
(* Group 2 *)                                       
OUT0200.CONFIG.SET_DIAG_LVL_PROT	(0, 2500, 100, eDIAG_PROT_MODE.DIAG_PROT);
OUT0201.CONFIG.SET_DIAG_LVL_PROT	(0, 2500, 100, eDIAG_PROT_MODE.DIAG_PROT);
OUT0202.CONFIG.SET_DIAG_LVL_PROT	(0, 2500, 100, eDIAG_PROT_MODE.DIAG_PROT);
OUT0203.CONFIG.SET_DIAG_LVL_PROT	(0, 2500, 100, eDIAG_PROT_MODE.DIAG_PROT);
OUT0204.CONFIG.SET_DIAG_LVL_PROT	(0, 2500, 100, eDIAG_PROT_MODE.DIAG_PROT);
OUT0205.CONFIG.SET_DIAG_LVL_PROT	(0, 2500, 100, eDIAG_PROT_MODE.DIAG_PROT);
OUT0206.CONFIG.SET_DIAG_LVL_PROT	(0, 4000, 100, eDIAG_PROT_MODE.DIAG_PROT);
OUT0207.CONFIG.SET_DIAG_LVL_PROT	(0, 4000, 100, eDIAG_PROT_MODE.DIAG_PROT);
OUT0208.CONFIG.SET_DIAG_LVL_PROT	(0, 4000, 100, eDIAG_PROT_MODE.DIAG_PROT);
END_ACTION

END_PROGRAM

// StandardPLC/Application/CAN_INIT
PROGRAM CAN_INIT
VAR
	xInit: BOOL:= TRUE;
	CAN0_Enable: ifmRCAN.CAN_Enable;
	CAN1_Enable: ifmRCAN.CAN_Enable;
	
END_VAR

IF xInit THEN
	
	CAN0_Enable(
	xEnable:= TRUE,
	echannel:= ifmDevice.CHAN_0,
	eBaudrate:= ifmDevice.KBAUD_250);
	CAN1_Enable(
	xEnable:= TRUE,
	eChannel:= ifmDevice.CHAN_1,
	eBaudrate:= ifmDevice.KBAUD_250);
	xInit:= FALSE;	
	
END_IF

END_PROGRAM

// StandardPLC/Application/CA_TX
PROGRAM CA_TX
VAR
	CAN_TX: ifmRCAN.CAN_TX;
	CANStatus:ifmRCAN.CAN_Status;
	aDATA: ARRAY[0..7] OF USINT:=[1,1,1,2,5,11,0];
	TON0: TON;
	TON_1: TON;
END_VAR

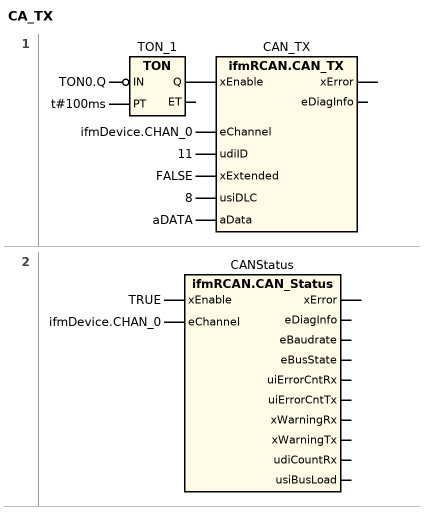
// NETWORK 1
TON_1(IN := NOT TON0.Q, PT := t#100ms); // TON
CAN_TX(
    xEnable := TON_1.Q,
    eChannel := ifmDevice.CHAN_0,
    udiID := 11,
    xExtended := FALSE,
    usiDLC := 8,
    aData := aDATA); // ifmRCAN.CAN_TX

// NETWORK 2
CANStatus(xEnable := TRUE, eChannel := ifmDevice.CHAN_0); // ifmRCAN.CAN_Status

END_PROGRAM

// StandardPLC/Application/CAN_RX
PROGRAM CAN_RX
VAR
	CAN_RX: ifmRCAN.CAN_RX;
	CANStatus: ifmRCAN.CAN_Status;
	aDATA: ARRAY [0..7] OF USINT;
END_VAR

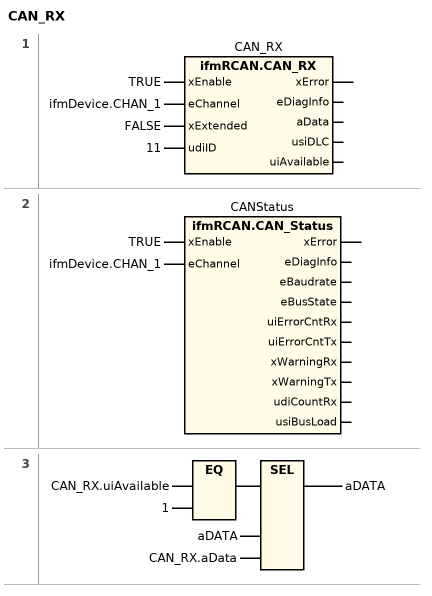
// NETWORK 1
CAN_RX(xEnable := TRUE, eChannel := ifmDevice.CHAN_1, xExtended := FALSE, udiID := 11); // ifmRCAN.CAN_RX

// NETWORK 2
CANStatus(xEnable := TRUE, eChannel := ifmDevice.CHAN_1); // ifmRCAN.CAN_Status

// NETWORK 3
aDATA := SEL(CAN_RX.uiAvailable = 1, aDATA, CAN_RX.aData);

END_PROGRAM
